(*

## Short summary
This interface provides assert statements for UTF-8 strings up to 255 bytes length

**Attention:** 
	All strings are handled as null-terminated byte streams

.. <legal notes>

legal notes
=================
| SPDX-FileCopyrightText: © 2024 ekvip automation GmbH <info@ekvip.de>
| SPDX-License-Identifier: Apache-2.0
| For details check: Apache-2.0_

.. _Apache-2.0: https://www.apache.org/licenses/LICENSE-2.0

.. </legal notes>



*)

INTERFACE IUtf8StringAssertions EXTENDS __SYSTEM.IQueryInterface

(*

## Short summary
This assertion method checks if the string ``stringToCheck`` contains the search string ``searchString``.
Processed strings must be in UTF-8 encoding

.. <legal notes>

legal notes
=================
| SPDX-FileCopyrightText: © 2024 ekvip automation GmbH <info@ekvip.de>
| SPDX-License-Identifier: Apache-2.0
| For details check: Apache-2.0_

.. _Apache-2.0: https://www.apache.org/licenses/LICENSE-2.0

.. </legal notes>



*)

METHOD contains
VAR_INPUT
	(* current string to check *)
	{attribute 'TcEncoding' := 'UTF-8'}
	stringToCheck	:Tc2_System.T_MaxString;
	(* string must be found in ``stringToCheck`` *)
	{attribute 'TcEncoding' := 'UTF-8'}
	searchString	:Tc2_System.T_MaxString;
	(* message if the assertion is false *)
	message			:AssertMessage;
	(* ``TRUE`` means ignore cases; ``FALSE`` means that cases must be equal too *)
	ignoreCases		:BOOL := FALSE;
	(*normalize both strings for check*)
	normalizeStrings :BOOL := TRUE;
END_VAR
END_METHOD

(*

## Short summary
This assertion method checks if the current string ``stringToCheck`` doesn't contain the search string ``searchString``.
Processed strings must be in UTF-8 encoding

.. <legal notes>

legal notes
=================
| SPDX-FileCopyrightText: © 2024 ekvip automation GmbH <info@ekvip.de>
| SPDX-License-Identifier: Apache-2.0
| For details check: Apache-2.0_

.. _Apache-2.0: https://www.apache.org/licenses/LICENSE-2.0

.. </legal notes>



*)

METHOD containsNo
VAR_INPUT
	(* current string to check *)
	{attribute 'TcEncoding' := 'UTF-8'}
	stringToCheck	:Tc2_System.T_MaxString;
	(* string that must not be found in ``stringToCheck`` *)
	{attribute 'TcEncoding' := 'UTF-8'}
	searchString	:Tc2_System.T_MaxString;
	(* message if the assertion is false *)
	message			:AssertMessage;
	(* ``TRUE`` means ignore cases; ``FALSE`` means that cases must be equal too *)
	ignoreCases		:BOOL := FALSE;
	(*normalize both strings for check*)
	normalizeStrings :BOOL := TRUE;
END_VAR
END_METHOD

(*

## Short summary
This assertion method checks if the current string ``stringToCheck`` ends with the string ``end``.
Processed strings must be in UTF-8 encoding

.. <legal notes>

legal notes
=================
| SPDX-FileCopyrightText: © 2024 ekvip automation GmbH <info@ekvip.de>
| SPDX-License-Identifier: Apache-2.0
| For details check: Apache-2.0_

.. _Apache-2.0: https://www.apache.org/licenses/LICENSE-2.0

.. </legal notes>



*)

METHOD endsWith
VAR_INPUT
	(* current string to check *)
	{attribute 'TcEncoding' := 'UTF-8'}
	stringToCheck	:Tc2_System.T_MaxString;
	(* expected end of ``stringToCheck`` *)
	{attribute 'TcEncoding' := 'UTF-8'}
	end				:Tc2_System.T_MaxString;
	(* message if the assertion is false *)
	message			:AssertMessage;
	(* ``TRUE`` means ignore cases; ``FALSE`` means that cases must be equal too *)
	ignoreCases		:BOOL := FALSE;
	(* ``TRUE`` means truncation of spaces on the right side of ``stringToCheck``*)
	trim		:BOOL := FALSE;
	(*normalize both strings for check*)
	normalizeStrings :BOOL := TRUE;
END_VAR
END_METHOD

(*

## Short summary
This assertion method checks if the current string ``stringToCheck`` is empty.
Processed strings must be in UTF-8 encoding

.. <legal notes>

legal notes
=================
| SPDX-FileCopyrightText: © 2024 ekvip automation GmbH <info@ekvip.de>
| SPDX-License-Identifier: Apache-2.0
| For details check: Apache-2.0_

.. _Apache-2.0: https://www.apache.org/licenses/LICENSE-2.0

.. </legal notes>



*)

METHOD isEmpty
VAR_INPUT
	(* current string to check *)
	{attribute 'TcEncoding' := 'UTF-8'}
	stringToCheck	:Tc2_System.T_MaxString;
	(* message if the assertion is false *)
	message			:AssertMessage;
END_VAR
END_METHOD

(*

## Short summary
This assertion method checks if the current string ``stringToCheck`` is equal to ``expected``.
Processed strings must be in UTF-8 encoding

.. <legal notes>

legal notes
=================
| SPDX-FileCopyrightText: © 2024 ekvip automation GmbH <info@ekvip.de>
| SPDX-License-Identifier: Apache-2.0
| For details check: Apache-2.0_

.. _Apache-2.0: https://www.apache.org/licenses/LICENSE-2.0

.. </legal notes>



*)

METHOD isEqualTo
VAR_INPUT
	(* current string to check *)
	{attribute 'TcEncoding' := 'UTF-8'}
	stringToCheck	:Tc2_System.T_MaxString;
	(* ``stringToCheck`` must be equal to expected *)
	{attribute 'TcEncoding' := 'UTF-8'}
	expected		:Tc2_System.T_MaxString;
	(* message if the assertion is false *)
	message			:AssertMessage;
	(* ``TRUE`` means ignore cases; ``FALSE`` means that cases must be equal too *)
	ignoreCases		:BOOL := FALSE;
	(*normalize both strings for check*)
	normalizeStrings :BOOL := TRUE;
END_VAR
END_METHOD

(*

## Short summary
This assertion method checks if the current string ``stringToCheck`` is not empty.
Processed strings must be in UTF-8 encoding

.. <legal notes>

legal notes
=================
| SPDX-FileCopyrightText: © 2024 ekvip automation GmbH <info@ekvip.de>
| SPDX-License-Identifier: Apache-2.0
| For details check: Apache-2.0_

.. _Apache-2.0: https://www.apache.org/licenses/LICENSE-2.0

.. </legal notes>



*)

METHOD isNotEmpty
VAR_INPUT
	(* current string to check *)
	{attribute 'TcEncoding' := 'UTF-8'}
	stringToCheck	:Tc2_System.T_MaxString;
	(* message if the assertion is false *)
	message			:AssertMessage;
END_VAR
END_METHOD

(*

## Short summary
This assertion method checks if the current string ``stringToCheck`` is not equal to ``unexpected``.
Processed strings must be in UTF-8 encoding

.. <legal notes>

legal notes
=================
| SPDX-FileCopyrightText: © 2024 ekvip automation GmbH <info@ekvip.de>
| SPDX-License-Identifier: Apache-2.0
| For details check: Apache-2.0_

.. _Apache-2.0: https://www.apache.org/licenses/LICENSE-2.0

.. </legal notes>



*)

METHOD isNotEqualTo
VAR_INPUT
	(* current string to check *)
	{attribute 'TcEncoding' := 'UTF-8'}
	stringToCheck	:Tc2_System.T_MaxString;
	(* ``stringToCheck`` must be not equal to expected *)
	{attribute 'TcEncoding' := 'UTF-8'}
	unexpected		:Tc2_System.T_MaxString;
	(* message if the assertion is false *)
	message			:AssertMessage;
	(* ``TRUE`` means ignore cases; ``FALSE`` means that cases must be equal too *)
	ignoreCases		:BOOL := FALSE;
	(*normalize both strings for check*)
	normalizeStrings :BOOL := TRUE;
END_VAR
END_METHOD

(*

## Short summary
This assertion method checks if the current string ``stringToCheck`` length is between ``minLength`` and ``maxLength``.
Processed strings must be in UTF-8 encoding

.. <legal notes>

legal notes
=================
| SPDX-FileCopyrightText: © 2024 ekvip automation GmbH <info@ekvip.de>
| SPDX-License-Identifier: Apache-2.0
| For details check: Apache-2.0_

.. _Apache-2.0: https://www.apache.org/licenses/LICENSE-2.0

.. </legal notes>



*)

METHOD lengthIsBetween
VAR_INPUT
	(* current string to check *)
	{attribute 'TcEncoding' := 'UTF-8'}
	stringToCheck		:Tc2_System.T_MaxString;
	(* lower limit of the string length *)
	minLength			:USINT;
	(* upper limit of the string length *)
	maxLength			:USINT;
	(* string length units of measurement *)
	stringLengthUnit	:UnicodeStringLengthUnit;
	(* message if the assertion is false *)
	message				:AssertMessage;
END_VAR
END_METHOD

(*

## Short summary
This assertion method checks if the current string ``stringToCheck`` length is equal to ``expectedLength``.
Processed strings must be in UTF-8 encoding

.. <legal notes>

legal notes
=================
| SPDX-FileCopyrightText: © 2024 ekvip automation GmbH <info@ekvip.de>
| SPDX-License-Identifier: Apache-2.0
| For details check: Apache-2.0_

.. _Apache-2.0: https://www.apache.org/licenses/LICENSE-2.0

.. </legal notes>



*)

METHOD lengthIsExact
VAR_INPUT
	(* current string to check *)
	{attribute 'TcEncoding' := 'UTF-8'}
	stringToCheck		:Tc2_System.T_MaxString;
	(* expected length of ``stringToCheck`` *)
	expectedLength		:USINT;
	(* string length units of measurement *)
	stringLengthUnit	:UnicodeStringLengthUnit;
	(* message if the assertion is false *)
	message				:AssertMessage;
END_VAR
END_METHOD

(*

## Short summary
This assertion method checks if the current string ``stringToCheck`` length is equal or less than to ``maxLength``.
Processed strings must be in UTF-8 encoding

.. <legal notes>

legal notes
=================
| SPDX-FileCopyrightText: © 2024 ekvip automation GmbH <info@ekvip.de>
| SPDX-License-Identifier: Apache-2.0
| For details check: Apache-2.0_

.. _Apache-2.0: https://www.apache.org/licenses/LICENSE-2.0

.. </legal notes>



*)

METHOD lengthIsMax
VAR_INPUT
	(* current string to check *)
	{attribute 'TcEncoding' := 'UTF-8'}
	stringToCheck		:Tc2_System.T_MaxString;
	(* upper limit of the length of ``stringToCheck`` *)
	maxLength			:USINT;
	(* string length units of measurement *)
	stringLengthUnit	:UnicodeStringLengthUnit;
	(* message if the assertion is false *)
	message				:AssertMessage;
END_VAR
END_METHOD

(*

## Short summary
This assertion method checks if the current string ``stringToCheck`` length is equal or grater than to ``minLength``.
Processed strings must be in UTF-8 encoding

.. <legal notes>

legal notes
=================
| SPDX-FileCopyrightText: © 2024 ekvip automation GmbH <info@ekvip.de>
| SPDX-License-Identifier: Apache-2.0
| For details check: Apache-2.0_

.. _Apache-2.0: https://www.apache.org/licenses/LICENSE-2.0

.. </legal notes>



*)

METHOD lengthIsMin
VAR_INPUT
	(* current string to check *)
	{attribute 'TcEncoding' := 'UTF-8'}
	stringToCheck		:Tc2_System.T_MaxString;
	(* lower limit of the length of ``stringToCheck`` *)
	minLength			:USINT;
	(* string length units of measurement *)
	stringLengthUnit	:UnicodeStringLengthUnit;
	(* message if the assertion is false *)
	message				:AssertMessage;
END_VAR
END_METHOD

(*

## Short summary
This assertion method checks if the current string ``stringToCheck`` starts with string ``start``.
Processed strings must be in UTF-8 encoding

.. <legal notes>

legal notes
=================
| SPDX-FileCopyrightText: © 2024 ekvip automation GmbH <info@ekvip.de>
| SPDX-License-Identifier: Apache-2.0
| For details check: Apache-2.0_

.. _Apache-2.0: https://www.apache.org/licenses/LICENSE-2.0

.. </legal notes>



*)

METHOD startsWith
VAR_INPUT
	(* current string to check *)
	{attribute 'TcEncoding' := 'UTF-8'}
	stringToCheck	:Tc2_System.T_MaxString;
	(* expected start of ``stringToCheck`` *)
	{attribute 'TcEncoding' := 'UTF-8'}
	start			:Tc2_System.T_MaxString;
	(* message if the assertion is false *)
	message			:AssertMessage;
	(* ``TRUE`` means ignore cases; ``FALSE`` means that cases must be equal too *)
	ignoreCases		:BOOL := FALSE;
	(* ``TRUE`` means truncation of spaces on the left side of ``stringToCheck``*)
	trim		:BOOL := FALSE;
	(*normalize both strings for check*)
	normalizeStrings :BOOL := TRUE;
END_VAR
END_METHOD

END_INTERFACE

(* stored: Version 1.1.0.1, ProductVersion 3.1.4026.11
   Itf IUtf8StringAssertions: Id {9ea562ca-dcb6-4825-96f6-da9541b09b54}
   Method contains: Id {896e8b99-bab7-4ded-aaa2-6faf60374597}
   Method containsNo: Id {0a87893a-c8f1-40fe-9f4e-30c135183624}
   Method endsWith: Id {9a59a8d8-9064-40c6-ae49-9860c4dc9bb9}
   Method isEmpty: Id {08345798-e89a-4dbb-bb31-bf39f0d618f8}
   Method isEqualTo: Id {ede01497-ae33-472d-8b32-8182d33e087f}
   Method isNotEmpty: Id {b5f155a7-3c15-4282-9b04-8cdff190382f}
   Method isNotEqualTo: Id {9779b346-dc67-4870-931b-1cdae18b98d7}
   Method lengthIsBetween: Id {e9aa007b-275a-4142-8f0f-4d1c7e939821}
   Method lengthIsExact: Id {270b0ced-aae6-49c3-8c01-0069c017efe8}
   Method lengthIsMax: Id {c4ced03e-8b11-4b04-b7fb-d283e820e4af}
   Method lengthIsMin: Id {4da1dd19-d6c9-4ab8-b36d-0ab5a6f1c595}
   Method startsWith: Id {e5dcf7f5-a4ae-4afe-a1fa-dfdd52997bfd} *)
